TYPE WrappedComponentExample_Config EXTENDS TcoCore.TcoStruct:
STRUCT

	VacuumReachedStabilisation:TIME:=T#100MS;
	VacuumPushTime:TIME:=T#100MS;
END_STRUCT
END_TYPE

(* stored: Version 1.1.0.1, ProductVersion 3.1.4024.12
   DUT WrappedComponentExample_Config: Id {fd4a1fe1-dfce-0359-2456-da059d207f84} *)
